SUBAPPLICATION Uebung_228_AX (* Ableitung von 227_AX: das Dreieck wird ROT außerhalb des Fensters -2..+2, GRÜN innerhalb *)
  (* Standard: 61499-2; Description: Copyright (c) 2026 Meisterschulen am Ostbahnhof This program and the accompanying materials are made available under the terms of the Eclipse Public License 2.0 which is available at https://www.eclipse.org/legal/epl-2.0/ SPDX-License-Identifier: EPL-2.0 *)
  (* Version 1.0, 2026-09-06, Franz Höpfinger, Meisterschulen am Ostbahnhof, initial API and implementation and/or initial documentation *)
  PACKAGE Uebungen;
  IMPORT Uebungen::const::UT::Dreieck::DefaultPool_Dreieck::FillStyle_Bargraph_Mittelmarker_Gruen;
  IMPORT Uebungen::const::UT::Dreieck::DefaultPool_Dreieck_PositionMarker::Container_PositionMarker;
  IMPORT Uebungen::const::UT::Dreieck::DefaultPool_Dreieck_BargraphSplit::Bargraph_Split_BargraphSplit;
  IMPORT Uebungen::const::UT::Dreieck::DefaultPool_Dreieck_Numeric::NumberVariable_Sollwert_N;
  IMPORT Uebungen::const::UT::Dreieck::DefaultPool_Dreieck_Numeric::NumberVariable_Istwert_N;
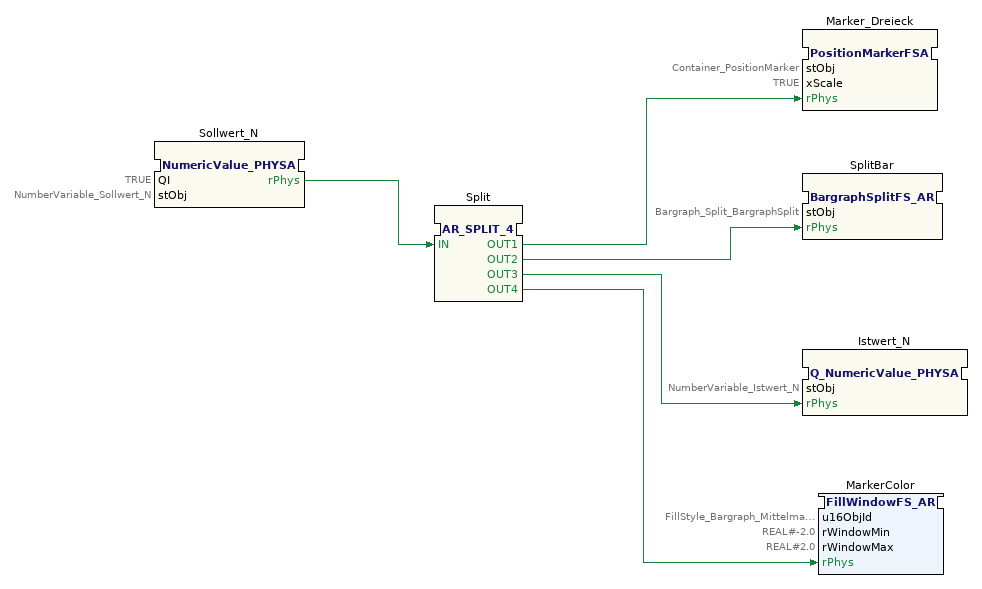
  FBS
    Sollwert_N : isobus::UT::io::NumericValue::NumericValue_PHYSA(QI := TRUE, stObj := NumberVariable_Sollwert_N);
    Split : adapter::events::unidirectional::AR_SPLIT_4;
    Marker_Dreieck : isobus::UT::Q::PositionMarkerFSA(stObj := Container_PositionMarker, xScale := TRUE);
    SplitBar : isobus::UT::Q::BargraphSplitFS_AR(stObj := Bargraph_Split_BargraphSplit);
    Istwert_N : isobus::UT::Q::Q_NumericValue_PHYSA(stObj := NumberVariable_Istwert_N);
  END_FBS
  SUBAPPS
    MarkerColor : MyLib::sys::FillWindowFS_AR(u16ObjId := FillStyle_Bargraph_Mittelmarker_Gruen, rWindowMin := REAL#-2.0, rWindowMax := REAL#2.0);
  END_SUBAPPS
  ADAPTER_CONNECTIONS
    Sollwert_N.rPhys TO Split.IN;
    Split.OUT1 TO Marker_Dreieck.rPhys;
    Split.OUT2 TO SplitBar.rPhys;
    Split.OUT3 TO Istwert_N.rPhys;
    Split.OUT4 TO MarkerColor.rPhys;
  END_CONNECTIONS
END_SUBAPPLICATION
